// TIA Portal V17 export
// export: Created 2022-05-07T16:02:26.3399099Z, ExportSetting WithDefaults, DisplayName Totally Integrated Automation Portal, DisplayVersion V17 Update 3, DisplayName TIA Portal Openness, DisplayVersion V17 Update 3, DisplayName TIA Portal Version Control Interface, DisplayVersion V17, DisplayName TIA Portal Test Suite Advanced, DisplayVersion V17 Update 1, DisplayName SINAMICS Startdrive Advanced, DisplayVersion V17 Update2, DisplayName SINAMICS Startdrive G130, G150, S120, S150, SINAMICS MV, S210, DisplayVersion V17 Update2, DisplayName SINAMICS Startdrive G110M, G120, G120C, G120D, G120P, G115D, DisplayVersion V17 Update2, DisplayName STEP 7 Professional, DisplayVersion V17 Update 3, DisplayName STEP 7 Safety, DisplayVersion V17, DisplayName WinCC UA Professional, DisplayVersion V17 Update 3
FUNCTION_BLOCK "CTRL_ASSE_STD"   // FB1, LAD
{ S7_Optimized_Access := 'TRUE' }
VERSION : 0.1
// FB STANDARD CONTROLLO ASSI
// stored: AutoNumber true, IsIECCheckEnabled false, IsRetainMemResEnabled false, MemoryReserve 100, SetENOAutomatically false, UDAEnableTagReadback false
   VAR_INPUT
      Automatico : Bool;
      Exe_MC_Reset : Bool;   // comando di reset
      En_MC_Power : Bool;   // abilitazione asse
      Exe_MC_Home : Bool;   // comando di homing
      Sp_Offset_Homing : Real;   // offset azzeramento
      Sp_Homing_Mode : Int;   // 0=diretto assoluto 2=passivo 3=attivo
      Exe_MC_Halt : Bool;   // comando HALT
      Exe_Jog_Fwd : Bool;   // comando jog +
      Exe_Jog_Bkw : Bool;   // comando jog -
      Sp_Jog_Velocity : Real;   // set velocità JOG
      Exe_MC_Velocity : Bool;   // comando velocità
      Sp_MC_Velocity : Real;   // set velocità Move Velocity
      Exe_MC_Relative : Bool;   // comando posizione relativa
      Sp_MoveRel_Distance : Real;   // set distanza Move Relative
      Sp_MoveRel_Velocity : Real;   // set velocità Move Relative
      Exe_MC_Abs : Bool;   // comando posizione assoluta
      Sp_MoveAbs_Position : Real;   // set posizione Move Absolute
      Sp_MoveAbs_Velocity : Real;   // set velocità Move Absolute
      Exe_MC_ChangeDyna : Bool;   // comando cambio dinamica
      Sp_RampUpTime : Real := 5.0;   // set tempo di rampa acc [s]
      Sp_RampDnTime : Real := 5.0;   // set tempo di rampa dec [s]
   END_VAR
   VAR_OUTPUT
      Output_MC_Reset_Done : Bool;   // asse resettato
      Output_MC_AxisEnabled : Bool;   // asse abilitato
      Output_MC_AxisHomed : Bool;   // asse homed (referenziato)
      Output_MC_Halt_Done : Bool;   // asse in halt
      Output_MC_JogInVelocity : Bool;   // vel raggiunta
      Output_MC_MoveInVelocity : Bool;   // vel raggiunta
      Output_MC_MoveRel_Done : Bool;   // move realtive eseguito
      Output_MC_MoveAbs_Done : Bool;   // move absolute eseguito
      Output_MC_MoveAbs_Busy : Bool;   // move absolute in corso
      Output_MC_At_Standstill : Bool;   // asse fermo
      Output_MC_Error : Bool;   // asse in errore (or di vari bool)
      Output_ActVelocity : Real;   // velocity attuale (asse)
      Output_ActPos : Real;   // posizione attuale
   END_VAR
   VAR_IN_OUT
      AxisTO : TO_PositioningAxis;
   END_VAR
   VAR
      AxisReady_PosAxis { S7_SetPoint := 'True'} : Bool;
      MC_Power_Instance { S7_SetPoint := 'True'} : MC_Power;
      MC_Reset_Instance { S7_SetPoint := 'True'} : MC_Reset;
      MC_Halt_Instance { S7_SetPoint := 'True'} : MC_Halt;
      MC_MoveJog_Instance { S7_SetPoint := 'True'} : MC_MoveJog;
      MC_MoveAbsolute_Instance { S7_SetPoint := 'True'} : MC_MoveAbsolute;
      MC_MoveVelocity_Instance { S7_SetPoint := 'True'} : MC_MoveVelocity;
      MC_Home_Instance { S7_SetPoint := 'True'} : MC_Home;
      MC_MoveRelative_Instance { S7_SetPoint := 'True'} : MC_MoveRelative;
      MC_ChangeDynamic_Instance { S7_SetPoint := 'True'} : MC_ChangeDynamic;
   END_VAR
BEGIN

REGION Network 1: MC_RESET
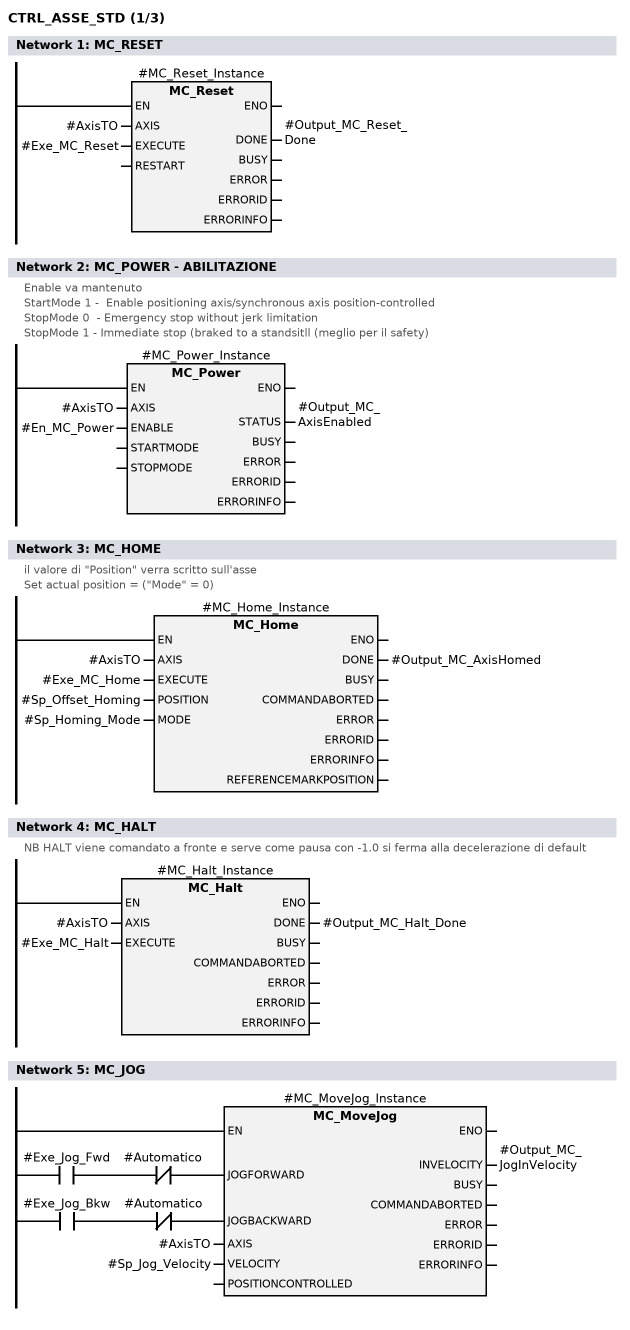
   RUNG wire#powerrail
      #MC_Reset_Instance.MC_Reset(Axis := #AxisTO, Execute := #Exe_MC_Reset, Restart :=, Done => #Output_MC_Reset_Done, Busy =>, Error =>, ErrorID =>, ErrorInfo =>)
   END_RUNG
   // the same network as SCL:
   #MC_Reset_Instance(Axis := #AxisTO, Execute := #Exe_MC_Reset, Done => #Output_MC_Reset_Done);   // MC_Reset
END_REGION

REGION Network 2: MC_POWER - ABILITAZIONE
   // Enable va mantenuto
   // StartMode 1 - ​​ Enable positioning axis/synchronous axis position-controlled
   // StopMode 0  - Emergency stop without jerk limitation
   // StopMode 1 - ​Immediate stop (braked to a standsitll (meglio per il safety)
   RUNG wire#powerrail
      #MC_Power_Instance.MC_Power(Axis := #AxisTO, Enable := #En_MC_Power, StartMode :=, StopMode :=, Status => #Output_MC_AxisEnabled, Busy =>, Error =>, ErrorID =>, ErrorInfo =>)
   END_RUNG
   // the same network as SCL:
   #MC_Power_Instance(Axis := #AxisTO, Enable := #En_MC_Power, Status => #Output_MC_AxisEnabled);   // MC_Power
END_REGION

REGION Network 3: MC_HOME
   // il valore di "Position" verra scritto sull'asse
   // Set actual position = ("Mode" = 0)
   RUNG wire#powerrail
      #MC_Home_Instance.MC_Home(Axis := #AxisTO, Execute := #Exe_MC_Home, Position := #Sp_Offset_Homing, Mode := #Sp_Homing_Mode, Done => #Output_MC_AxisHomed, Busy =>, CommandAborted =>, Error =>, ErrorID =>, ErrorInfo =>, ReferenceMarkPosition =>)
   END_RUNG
   // the same network as SCL:
   #MC_Home_Instance(Axis := #AxisTO,   // MC_Home
                     Execute := #Exe_MC_Home,
                     Position := #Sp_Offset_Homing,
                     Mode := #Sp_Homing_Mode,
                     Done => #Output_MC_AxisHomed);
END_REGION

REGION Network 4: MC_HALT
   // NB HALT viene comandato a fronte e serve come pausa con -1.0 si ferma alla decelerazione di default
   RUNG wire#powerrail
      #MC_Halt_Instance.MC_Halt(Axis := #AxisTO, Execute := #Exe_MC_Halt, Done => #Output_MC_Halt_Done, Busy =>, CommandAborted =>, Error =>, ErrorID =>, ErrorInfo =>)
   END_RUNG
   // the same network as SCL:
   #MC_Halt_Instance(Axis := #AxisTO, Execute := #Exe_MC_Halt, Done => #Output_MC_Halt_Done);   // MC_Halt
END_REGION

REGION Network 5: MC_JOG
   RUNG wire#powerrail
      #MC_MoveJog_Instance.MC_MoveJog(JogForward := wire#w1, JogBackward := wire#w2, Axis := #AxisTO, Velocity := #Sp_Jog_Velocity, PositionControlled :=, InVelocity => #Output_MC_JogInVelocity, Busy =>, CommandAborted =>, Error =>, ErrorID =>, ErrorInfo =>)
   END_RUNG
   RUNG wire#powerrail
      Contact( #Exe_Jog_Fwd )
      I_Contact( #Automatico )
   END_RUNG wire#w1
   RUNG wire#powerrail
      Contact( #Exe_Jog_Bkw )
      I_Contact( #Automatico )
   END_RUNG wire#w2
   // the same network as SCL:
   #MC_MoveJog_Instance(JogForward := #Exe_Jog_Fwd AND NOT #Automatico,   // MC_MoveJog
                        JogBackward := #Exe_Jog_Bkw AND NOT #Automatico,
                        Axis := #AxisTO,
                        Velocity := #Sp_Jog_Velocity,
                        InVelocity => #Output_MC_JogInVelocity);
END_REGION

REGION Network 6: MC_VELOCITY
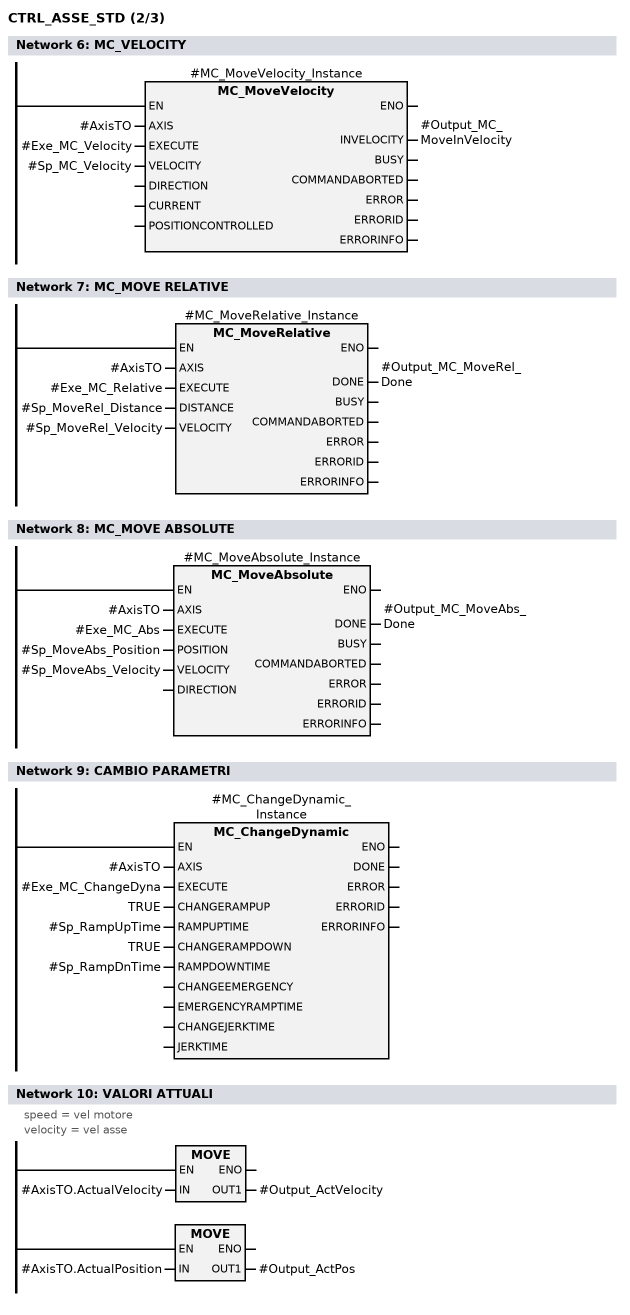
   RUNG wire#powerrail
      #MC_MoveVelocity_Instance.MC_MoveVelocity(Axis := #AxisTO, Execute := #Exe_MC_Velocity, Velocity := #Sp_MC_Velocity, Direction :=, Current :=, PositionControlled :=, InVelocity => #Output_MC_MoveInVelocity, Busy =>, CommandAborted =>, Error =>, ErrorID =>, ErrorInfo =>)
   END_RUNG
   // the same network as SCL:
   #MC_MoveVelocity_Instance(Axis := #AxisTO,   // MC_MoveVelocity
                           Execute := #Exe_MC_Velocity,
                           Velocity := #Sp_MC_Velocity,
                           InVelocity => #Output_MC_MoveInVelocity);
END_REGION

REGION Network 7: MC_MOVE RELATIVE
   RUNG wire#powerrail
      #MC_MoveRelative_Instance.MC_MoveRelative(Axis := #AxisTO, Execute := #Exe_MC_Relative, Distance := #Sp_MoveRel_Distance, Velocity := #Sp_MoveRel_Velocity, Done => #Output_MC_MoveRel_Done, Busy =>, CommandAborted =>, Error =>, ErrorID =>, ErrorInfo =>)
   END_RUNG
   // the same network as SCL:
   #MC_MoveRelative_Instance(Axis := #AxisTO,   // MC_MoveRelative
                           Execute := #Exe_MC_Relative,
                           Distance := #Sp_MoveRel_Distance,
                           Velocity := #Sp_MoveRel_Velocity,
                           Done => #Output_MC_MoveRel_Done);
END_REGION

REGION Network 8: MC_MOVE ABSOLUTE
   RUNG wire#powerrail
      #MC_MoveAbsolute_Instance.MC_MoveAbsolute(Axis := #AxisTO, Execute := #Exe_MC_Abs, Position := #Sp_MoveAbs_Position, Velocity := #Sp_MoveAbs_Velocity, Direction :=, Done => #Output_MC_MoveAbs_Done, Busy =>, CommandAborted =>, Error =>, ErrorID =>, ErrorInfo =>)
   END_RUNG
   // the same network as SCL:
   #MC_MoveAbsolute_Instance(Axis := #AxisTO,   // MC_MoveAbsolute
                           Execute := #Exe_MC_Abs,
                           Position := #Sp_MoveAbs_Position,
                           Velocity := #Sp_MoveAbs_Velocity,
                           Done => #Output_MC_MoveAbs_Done);
END_REGION

REGION Network 9: CAMBIO PARAMETRI
   RUNG wire#powerrail
      #MC_ChangeDynamic_Instance.MC_ChangeDynamic(Axis := #AxisTO, Execute := #Exe_MC_ChangeDyna, ChangeRampUp := TRUE, RampUpTime := #Sp_RampUpTime, ChangeRampDown := TRUE, RampDownTime := #Sp_RampDnTime, ChangeEmergency :=, EmergencyRampTime :=, ChangeJerkTime :=, JerkTime :=, Done =>, Error =>, ErrorID =>, ErrorInfo =>)
   END_RUNG
   // the same network as SCL:
   #MC_ChangeDynamic_Instance(Axis := #AxisTO,   // MC_ChangeDynamic
                           Execute := #Exe_MC_ChangeDyna,
                           ChangeRampUp := TRUE,
                           RampUpTime := #Sp_RampUpTime,
                           ChangeRampDown := TRUE,
                           RampDownTime := #Sp_RampDnTime);
END_REGION

REGION Network 10: VALORI ATTUALI
   // speed = vel motore 
   // velocity = vel asse
   RUNG wire#powerrail
      Move(in := #AxisTO.ActualVelocity, out1 => #Output_ActVelocity)
   END_RUNG
   RUNG wire#powerrail
      Move(in := #AxisTO.ActualPosition, out1 => #Output_ActPos)
   END_RUNG
   // the same network as SCL:
   #Output_ActVelocity := #AxisTO.ActualVelocity;
   #Output_ActPos := #AxisTO.ActualPosition;
END_REGION

REGION Network 11: STANDSTILL
   // VERIFICARE VELOCITA' A ZERO
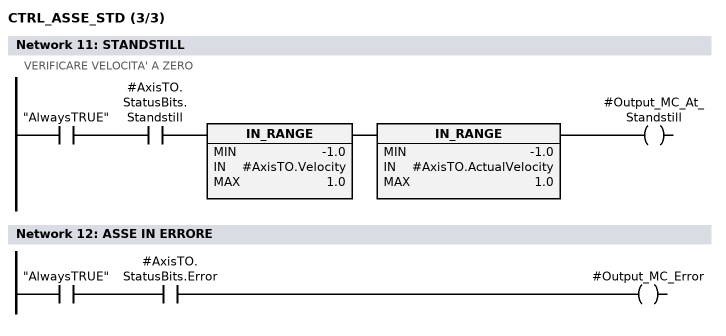
   RUNG wire#powerrail
      Contact( "AlwaysTRUE" )
      Contact( #AxisTO.StatusBits.Standstill )
      { S7_Templates := "SrcType := Real" } InRange(min := -1.0, in := #AxisTO.Velocity, max := 1.0)
      { S7_Templates := "SrcType := LReal" } InRange(min := -1.0, in := #AxisTO.ActualVelocity, max := 1.0)
      Coil( #Output_MC_At_Standstill )
   END_RUNG
   // the same network as SCL:
   #Output_MC_At_Standstill := "AlwaysTRUE" AND #AxisTO.StatusBits.Standstill AND (-1.0 <= #AxisTO.Velocity) AND (#AxisTO.Velocity <= 1.0) AND (-1.0 <= #AxisTO.ActualVelocity) AND (#AxisTO.ActualVelocity <= 1.0);
END_REGION

REGION Network 12: ASSE IN ERRORE
   RUNG wire#powerrail
      Contact( "AlwaysTRUE" )
      Contact( #AxisTO.StatusBits.Error )
      Coil( #Output_MC_Error )
   END_RUNG
   // the same network as SCL:
   #Output_MC_Error := "AlwaysTRUE" AND #AxisTO.StatusBits.Error;
END_REGION
END_FUNCTION_BLOCK
